// TIA Portal V19 export
TYPE "Coil_Item"
// stored: Access Published
   STRUCT
      C_ID : DInt;   // Coil ID
      MES_IDP : String;
      Decoiler_N : Int;   // Rotolo su Aspo 1 / 2
      MES_CN : String;   // [MES_CN] Numero identificativo del rotolo
      MES_HN : String;   // [MES_HN] Numero di colata
      Stato_Rotolo : Int;   // [MES_SR] Stao rotolo: 0=Vuoto; 1=In uso; 2=Fine lamiera; 3=Interruzione
      Provini_Richiesti : Int;   // [MES_PPR] Provini richiesti
      Provini_Eseguiti : Int;   // [MES_PRD] Provini eseguiti
      Diametro_Rotolo : Real;   // [MES_RDM] Diametro rotolo
      Spessore_Errore : Int;   // [MES_TNG] Presenza errore spessore: 0 = No; >=1 = Si
      Spessore_materiale_TAV : Real;   // [MES_TAV] Valore spessore letto dal sensore (in mm)
      Spessore_materiale_TEV : Real;   // [MES_TEV] Valore fuori tolleranza (in mm)
      Spessore_Deroga_TKD : Int;   // [MES_TKD] Uso del rotolo “in deroga” nonostante la presenza di errore spessore ([TNG] ≥ 1)
   END_STRUCT;
END_TYPE
